// TIA Portal V20 export
TYPE "LBP_typeTMLoadMT"
TITLE = Tool management / Gestion des outils
// User data type for block LBP_TMLoadMT [DB1071] / Type de données utilisateur pour bloc LBP_TMLoadMT [DB1071]
   STRUCT
      MTIF : Array[1..16] of Struct
         DistanceCoding : Int;   // Type of distance coding ($TC_MTP_KD) / Type de codage de distance ($TC_MTP_KD)
         Places : Int;   // Number of locations of the multitool / Nombre d'emplacements Multitool
         Distance : Real;   // Multitool location distance / Distance de l'emplacement Multitool
         MTNo : Int;   // Internal T number of the multitool / Numéro d'outil interne du Multitool
         PlaceNo : Int;   // Location number within the multitool to which the system positions / Numéro d'emplacement Multitool cible de positionnement du système
         Toolholder : Int;   // Spindle or toolholder number / Numéro de broche ou porte-outil
         reserved : Array[1..3] of Int;   // Reserved / Réservé
      END_STRUCT;
   END_STRUCT;
   // // MTIF[2].DistanceCoding : Type of distance coding ($TC_MTP_KD) / Type de codage de distance ($TC_MTP_KD)
   // // MTIF[3].DistanceCoding : Type of distance coding ($TC_MTP_KD) / Type de codage de distance ($TC_MTP_KD)
   // // MTIF[4].DistanceCoding : Type of distance coding ($TC_MTP_KD) / Type de codage de distance ($TC_MTP_KD)
   // // MTIF[5].DistanceCoding : Type of distance coding ($TC_MTP_KD) / Type de codage de distance ($TC_MTP_KD)
   // // MTIF[6].DistanceCoding : Type of distance coding ($TC_MTP_KD) / Type de codage de distance ($TC_MTP_KD)
   // // MTIF[7].DistanceCoding : Type of distance coding ($TC_MTP_KD) / Type de codage de distance ($TC_MTP_KD)
   // // MTIF[8].DistanceCoding : Type of distance coding ($TC_MTP_KD) / Type de codage de distance ($TC_MTP_KD)
   // // MTIF[9].DistanceCoding : Type of distance coding ($TC_MTP_KD) / Type de codage de distance ($TC_MTP_KD)
   // // MTIF[10].DistanceCoding : Type of distance coding ($TC_MTP_KD) / Type de codage de distance ($TC_MTP_KD)
   // // MTIF[11].DistanceCoding : Type of distance coding ($TC_MTP_KD) / Type de codage de distance ($TC_MTP_KD)
   // // MTIF[12].DistanceCoding : Type of distance coding ($TC_MTP_KD) / Type de codage de distance ($TC_MTP_KD)
   // // MTIF[13].DistanceCoding : Type of distance coding ($TC_MTP_KD) / Type de codage de distance ($TC_MTP_KD)
   // // MTIF[14].DistanceCoding : Type of distance coding ($TC_MTP_KD) / Type de codage de distance ($TC_MTP_KD)
   // // MTIF[15].DistanceCoding : Type of distance coding ($TC_MTP_KD) / Type de codage de distance ($TC_MTP_KD)
   // // MTIF[16].DistanceCoding : Type of distance coding ($TC_MTP_KD) / Type de codage de distance ($TC_MTP_KD)
   // // MTIF[2].Places : Number of locations of the multitool / Nombre d'emplacements Multitool
   // // MTIF[3].Places : Number of locations of the multitool / Nombre d'emplacements Multitool
   // // MTIF[4].Places : Number of locations of the multitool / Nombre d'emplacements Multitool
   // // MTIF[5].Places : Number of locations of the multitool / Nombre d'emplacements Multitool
   // // MTIF[6].Places : Number of locations of the multitool / Nombre d'emplacements Multitool
   // // MTIF[7].Places : Number of locations of the multitool / Nombre d'emplacements Multitool
   // // MTIF[8].Places : Number of locations of the multitool / Nombre d'emplacements Multitool
   // // MTIF[9].Places : Number of locations of the multitool / Nombre d'emplacements Multitool
   // // MTIF[10].Places : Number of locations of the multitool / Nombre d'emplacements Multitool
   // // MTIF[11].Places : Number of locations of the multitool / Nombre d'emplacements Multitool
   // // MTIF[12].Places : Number of locations of the multitool / Nombre d'emplacements Multitool
   // // MTIF[13].Places : Number of locations of the multitool / Nombre d'emplacements Multitool
   // // MTIF[14].Places : Number of locations of the multitool / Nombre d'emplacements Multitool
   // // MTIF[15].Places : Number of locations of the multitool / Nombre d'emplacements Multitool
   // // MTIF[16].Places : Number of locations of the multitool / Nombre d'emplacements Multitool
   // // MTIF[2].Distance : Multitool location distance / Distance de l'emplacement Multitool
   // // MTIF[3].Distance : Multitool location distance / Distance de l'emplacement Multitool
   // // MTIF[4].Distance : Multitool location distance / Distance de l'emplacement Multitool
   // // MTIF[5].Distance : Multitool location distance / Distance de l'emplacement Multitool
   // // MTIF[6].Distance : Multitool location distance / Distance de l'emplacement Multitool
   // // MTIF[7].Distance : Multitool location distance / Distance de l'emplacement Multitool
   // // MTIF[8].Distance : Multitool location distance / Distance de l'emplacement Multitool
   // // MTIF[9].Distance : Multitool location distance / Distance de l'emplacement Multitool
   // // MTIF[10].Distance : Multitool location distance / Distance de l'emplacement Multitool
   // // MTIF[11].Distance : Multitool location distance / Distance de l'emplacement Multitool
   // // MTIF[12].Distance : Multitool location distance / Distance de l'emplacement Multitool
   // // MTIF[13].Distance : Multitool location distance / Distance de l'emplacement Multitool
   // // MTIF[14].Distance : Multitool location distance / Distance de l'emplacement Multitool
   // // MTIF[15].Distance : Multitool location distance / Distance de l'emplacement Multitool
   // // MTIF[16].Distance : Multitool location distance / Distance de l'emplacement Multitool
   // // MTIF[2].MTNo : Internal T number of the multitool / Numéro d'outil interne du Multitool
   // // MTIF[3].MTNo : Internal T number of the multitool / Numéro d'outil interne du Multitool
   // // MTIF[4].MTNo : Internal T number of the multitool / Numéro d'outil interne du Multitool
   // // MTIF[5].MTNo : Internal T number of the multitool / Numéro d'outil interne du Multitool
   // // MTIF[6].MTNo : Internal T number of the multitool / Numéro d'outil interne du Multitool
   // // MTIF[7].MTNo : Internal T number of the multitool / Numéro d'outil interne du Multitool
   // // MTIF[8].MTNo : Internal T number of the multitool / Numéro d'outil interne du Multitool
   // // MTIF[9].MTNo : Internal T number of the multitool / Numéro d'outil interne du Multitool
   // // MTIF[10].MTNo : Internal T number of the multitool / Numéro d'outil interne du Multitool
   // // MTIF[11].MTNo : Internal T number of the multitool / Numéro d'outil interne du Multitool
   // // MTIF[12].MTNo : Internal T number of the multitool / Numéro d'outil interne du Multitool
   // // MTIF[13].MTNo : Internal T number of the multitool / Numéro d'outil interne du Multitool
   // // MTIF[14].MTNo : Internal T number of the multitool / Numéro d'outil interne du Multitool
   // // MTIF[15].MTNo : Internal T number of the multitool / Numéro d'outil interne du Multitool
   // // MTIF[16].MTNo : Internal T number of the multitool / Numéro d'outil interne du Multitool
   // // MTIF[2].PlaceNo : Location number within the multitool to which the system positions / Numéro d'emplacement Multitool cible de positionnement du système
   // // MTIF[3].PlaceNo : Location number within the multitool to which the system positions / Numéro d'emplacement Multitool cible de positionnement du système
   // // MTIF[4].PlaceNo : Location number within the multitool to which the system positions / Numéro d'emplacement Multitool cible de positionnement du système
   // // MTIF[5].PlaceNo : Location number within the multitool to which the system positions / Numéro d'emplacement Multitool cible de positionnement du système
   // // MTIF[6].PlaceNo : Location number within the multitool to which the system positions / Numéro d'emplacement Multitool cible de positionnement du système
   // // MTIF[7].PlaceNo : Location number within the multitool to which the system positions / Numéro d'emplacement Multitool cible de positionnement du système
   // // MTIF[8].PlaceNo : Location number within the multitool to which the system positions / Numéro d'emplacement Multitool cible de positionnement du système
   // // MTIF[9].PlaceNo : Location number within the multitool to which the system positions / Numéro d'emplacement Multitool cible de positionnement du système
   // // MTIF[10].PlaceNo : Location number within the multitool to which the system positions / Numéro d'emplacement Multitool cible de positionnement du système
   // // MTIF[11].PlaceNo : Location number within the multitool to which the system positions / Numéro d'emplacement Multitool cible de positionnement du système
   // // MTIF[12].PlaceNo : Location number within the multitool to which the system positions / Numéro d'emplacement Multitool cible de positionnement du système
   // // MTIF[13].PlaceNo : Location number within the multitool to which the system positions / Numéro d'emplacement Multitool cible de positionnement du système
   // // MTIF[14].PlaceNo : Location number within the multitool to which the system positions / Numéro d'emplacement Multitool cible de positionnement du système
   // // MTIF[15].PlaceNo : Location number within the multitool to which the system positions / Numéro d'emplacement Multitool cible de positionnement du système
   // // MTIF[16].PlaceNo : Location number within the multitool to which the system positions / Numéro d'emplacement Multitool cible de positionnement du système
   // // MTIF[2].Toolholder : Spindle or toolholder number / Numéro de broche ou porte-outil
   // // MTIF[3].Toolholder : Spindle or toolholder number / Numéro de broche ou porte-outil
   // // MTIF[4].Toolholder : Spindle or toolholder number / Numéro de broche ou porte-outil
   // // MTIF[5].Toolholder : Spindle or toolholder number / Numéro de broche ou porte-outil
   // // MTIF[6].Toolholder : Spindle or toolholder number / Numéro de broche ou porte-outil
   // // MTIF[7].Toolholder : Spindle or toolholder number / Numéro de broche ou porte-outil
   // // MTIF[8].Toolholder : Spindle or toolholder number / Numéro de broche ou porte-outil
   // // MTIF[9].Toolholder : Spindle or toolholder number / Numéro de broche ou porte-outil
   // // MTIF[10].Toolholder : Spindle or toolholder number / Numéro de broche ou porte-outil
   // // MTIF[11].Toolholder : Spindle or toolholder number / Numéro de broche ou porte-outil
   // // MTIF[12].Toolholder : Spindle or toolholder number / Numéro de broche ou porte-outil
   // // MTIF[13].Toolholder : Spindle or toolholder number / Numéro de broche ou porte-outil
   // // MTIF[14].Toolholder : Spindle or toolholder number / Numéro de broche ou porte-outil
   // // MTIF[15].Toolholder : Spindle or toolholder number / Numéro de broche ou porte-outil
   // // MTIF[16].Toolholder : Spindle or toolholder number / Numéro de broche ou porte-outil
   // // MTIF[2].reserved : Reserved / Réservé
   // // MTIF[3].reserved : Reserved / Réservé
   // // MTIF[4].reserved : Reserved / Réservé
   // // MTIF[5].reserved : Reserved / Réservé
   // // MTIF[6].reserved : Reserved / Réservé
   // // MTIF[7].reserved : Reserved / Réservé
   // // MTIF[8].reserved : Reserved / Réservé
   // // MTIF[9].reserved : Reserved / Réservé
   // // MTIF[10].reserved : Reserved / Réservé
   // // MTIF[11].reserved : Reserved / Réservé
   // // MTIF[12].reserved : Reserved / Réservé
   // // MTIF[13].reserved : Reserved / Réservé
   // // MTIF[14].reserved : Reserved / Réservé
   // // MTIF[15].reserved : Reserved / Réservé
   // // MTIF[16].reserved : Reserved / Réservé
END_TYPE
